{attribute 'qualified_only'}
VAR_GLOBAL
	GrindingWheelMS AT %Q* : BOOL;
	StartGrindingWheelPB AT %I* : BOOL;
	StopGrindingWheelPB AT %I* : BOOL;
END_VAR

(* stored: Version 1.1.0.1, ProductVersion 3.1.4024.12
   GVL GVL_Grinding: Id {b5db8d1c-63aa-412a-b4aa-18b564493082} *)
